FUNCTION_BLOCK FB_mbReadRobotTaskStatusInfo
VAR_INPUT
	Robot : STRING;
END_VAR
VAR_OUTPUT
	stTaskStatusInfo : ST_RobotTaskStatusInfo;
END_VAR
VAR
	Value : ARRAY [1..12] OF WORD;
	mbRead : FB_mbReadRegs;
	state : int;
END_VAR

(* 
FB_mbReadRobotStatusInfo - Function Block that can be called to read a Robot status registers: 128-139
	INPUTS:
		- Robot : Sting, 'UR5' or 'UR3'
	OUTPUTS
		- RobotTaskStatus : WORD;
		- ZoneOccupied : WORD;
		- IsInTask : BOOL;
		- IsPerformingTaskAction : BOOL;
*)

// Set function block vairables
mbRead.nQuantity := 12;
mbRead.cbLength := 24;

IF Robot='UR5' THEN
	mbRead.sIPAddr := Global.stUR5.IP;
	mbRead.nTCPPort := Global.stUR5.mbPort;
	mbRead.nUnitID := Global.stUR5.unitID;
ELSIF Robot='UR3' THEN
	mbRead.sIPAddr := Global.stUR3.IP;
	mbRead.nTCPPort := Global.stUR3.mbPort;
	mbRead.nUnitID := Global.stUR3.unitID;
END_IF

mbRead.pDestAddr := ADR(Value);
mbRead.nMBAddr := 128;

// Set/Determine State of Function block
CASE state OF
	0:
		mbRead.bExecute := TRUE;
		state := 10;
	10:
		IF NOT mbRead.bBusy THEN
			mbRead.bExecute :=FALSE;
			state := 20;
		END_IF
	20:
		stTaskStatusInfo.nRobotTaskStatus := Value[1];
		stTaskStatusInfo.nZoneOccupied := Value[2];
		stTaskStatusInfo.bInTask := INT_TO_BOOL(Value[3]);
		stTaskStatusInfo.bPerformingTaskAction := INT_TO_BOOL(Value[4]);
		
		IF stTaskStatusInfo.nRobotTaskStatus = 1 THEN
			stTaskStatusInfo.sRobotStatus := 'Waiting for Task Assignment';
		ELSIF stTaskStatusInfo.nRobotTaskStatus = 2 THEN
			stTaskStatusInfo.sRobotStatus := 'Executing Assigned Task';
		END_IF

		state := 0;
END_CASE

// Run function block
mbRead();

END_FUNCTION_BLOCK

(* stored: Version 1.1.0.1, ProductVersion 3.1.4020.12
   POU FB_mbReadRobotTaskStatusInfo: Id {fefaa6e2-e81f-4ae4-b48c-1980aeba3e13}, SpecialFunc None *)
